FUNCTION_BLOCK FB_PepperoniPizza EXTENDS FB_Pizza
VAR_INPUT
END_VAR
VAR_OUTPUT
END_VAR
VAR
END_VAR

METHOD addCheese
VAR_INPUT
END_VAR
ADSLOGSTR( msgCtrlMask := ADSLOG_MSGTYPE_WARN,
        	msgFmtStr := 'Adding Mozzarella Cheese...', '');
END_METHOD

METHOD addMeat
VAR_INPUT
END_VAR
ADSLOGSTR( msgCtrlMask := ADSLOG_MSGTYPE_WARN,
        	msgFmtStr := 'Adding Pepperoni...', '');
END_METHOD

METHOD addVegetables : BOOL
VAR_INPUT
END_VAR
// Nothing here because it's not used
// Normally these Meat, Cheese, and Veg would be an Abstract Method
END_METHOD

METHOD customerWantsCheese : BOOL
VAR_INPUT
END_VAR
// Cheese Hook
customerWantsCheese := TRUE;
END_METHOD

METHOD customerWantsMeat : BOOL
VAR_INPUT
END_VAR
// Meat Hook
customerWantsMeat := TRUE;
END_METHOD

END_FUNCTION_BLOCK

(* stored: Version 1.1.0.1, ProductVersion 3.1.4024.12
   POU FB_PepperoniPizza: Id {0eb8e661-ef29-4055-9860-b4646f7eb3a1}, SpecialFunc None
   Method addCheese: Id {bcbcec8e-55a0-481b-aa1d-e1a090df105f}
   Method addMeat: Id {411ea7c7-d2cd-45a6-9023-bc48d40ecf58}
   Method addVegetables: Id {95337c26-1b6b-4834-a857-b0f543048b9e}
   Method customerWantsCheese: Id {59e799b7-c0fb-43f9-ad82-197750dcba5f}
   Method customerWantsMeat: Id {19909c54-d593-42fe-8e86-9689eda1c885} *)
